// Sets the boolean value to true if it is false and returns true if it was false before being set.
FUNCTION F_SetOnFalse : BOOL // Whether the value was false before setting.
VAR_INPUT
    bValue : REFERENCE TO BOOL; // Boolean value to set.
END_VAR

F_SetOnFalse 	:= NOT bValue;
bValue 			:= TRUE;

END_FUNCTION

(* stored: Version 1.1.0.1
   POU F_SetOnFalse: Id {e0f7f683-639f-0a70-0cc8-f72bf13e651c}, SpecialFunc None *)
